{attribute 'qualified_only'}
{attribute 'strict'}
TYPE E_HmiLanguage :
(
	English 	:= 1,
	Mandarin 	:= 2,
	German 		:= 3,
	French 		:= 4,
	Portuguese 	:= 5
);
END_TYPE

(* stored: Version 1.1.0.1, ProductVersion 3.1.4024.12
   DUT E_HmiLanguage: Id {94bab743-3117-469f-8582-251742093805} *)
